# B&R Automation Studio project PLC_base3
Automation Studio 4.8.2.72

## Configuration Config1

CPU X20CP1382, AutomationRuntime B4.82, Build 4.1.2, Vc V4.72.1

### IoMap.iom - X20CP1382/IoMap.iom
```iecst
VAR_CONFIG
	::Program:enable1 AT %QX."X3a".DigitalOutput01;
	::Program:enable2 AT %QX."X3a".DigitalOutput02;
	::Program:enable3 AT %QX."X3a".DigitalOutput03;
	::Program:direction1 AT %QX."X3a".DigitalOutput04;
	::Program:direction2 AT %QX."X3a".DigitalOutput05;
	::Program:direction3 AT %QX."X3a".DigitalOutput06;
	::Program:bspidser AT %QX."X3a".DigitalOutput08;
	::Program:step1x AT %QX."X3a".DigitalOutput09;
	::Program:step2y AT %QX."X3a".DigitalOutput10;
	::Program:step3z AT %QX."X3a".DigitalOutput11;
	::Program:stop3 AT %IX."X1a".DigitalInput01;
	::Program:stop2 AT %IX."X1a".DigitalInput02;
	::Program:stop1 AT %IX."X1a".DigitalInput03;
	::Program:stopb AT %IX."X1a".DigitalInput04;
END_VAR
```

## Logical view

Binary libraries used (declarations not repeated): AsIecCon

### Program Logical/Program (IEC)

#### Main.st - Init, cyclic, exit code
```iecst
PROGRAM _INIT
	enable1 := FALSE;
	enable2 := FALSE;
	enable3 := FALSE;

count:= 0;

END_PROGRAM

PROGRAM _CYCLIC
(*	IF   start1 = TRUE THEN

		IF stop3 = FALSE AND stop1 = FALSE THEN
			direction3 := FALSE;
	  		step3z := NOT step3z;
		END_IF;

		IF stop1 = FALSE AND stop3 = TRUE THEN
			(*IF step1x = FALSE THEN
				step1x := TRUE;
			ELSIF
				step1x = TRUE THEN
				step1x := FALSE;

			END_IF;*)
	    (*	step1x := NOT step1x;
		END_IF;

		IF stopb = FALSE AND stop1 = TRUE THEN
			direction3 := TRUE;
			step3z := NOT step3z;
		END_IF;*)
(*
		timer.IN := NOT timer.Q;
		timer.PT := T#5s;
		timer();
		bspidser := timer.Q;
(*
		IF stop3 = FALSE THEN
			direction3 := FALSE;
			step3z := NOT step3z;
		END_IF;

		//mynikkr

	END_IF;*)
	IF start1 = TRUE THEN

	IF stop1 = FALSE THEN
			step1x := NOT step1x;
			count := count + 1;
	END_IF

		IF stop1 = TRUE THEN
	  start1 := FALSE;
		END_IF;

	END_IF;

END_PROGRAM

PROGRAM _EXIT
	(* Insert code here *)

END_PROGRAM
```

#### Variables.var - Local variables
```iecst
VAR
	count : UINT;
	bspidser : {REDUND_UNREPLICABLE} BOOL;
	enable1 : {REDUND_UNREPLICABLE} BOOL;
	enable2 : {REDUND_UNREPLICABLE} BOOL;
	enable3 : {REDUND_UNREPLICABLE} BOOL;
	direction1 : BOOL;
	direction2 : BOOL;
	direction3 : BOOL;
	step1x : BOOL;
	step2y : BOOL;
	step3z : BOOL;
	stopb : BOOL;
	stop1 : BOOL;
	stop2 : BOOL;
	stop3 : BOOL;
	start1 : BOOL;
	timer : TON;
END_VAR
```

Listed in the project but not available here: Logical/Program/Types.typ
